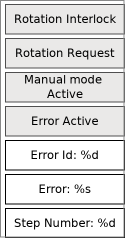
VISUALIZATION vTableBaseStationInfo  // 125x238
VAR_IN_OUT
	fbStation:FB_BaseStation;
END_VAR
    Rectangle (5,38 120x30), "Rotation Request", colour toggle: fbStation.bRotationRequest
    Rectangle (5,4 120x30), "Rotation Interlock", colour toggle: fbStation.bRotationInterlock
    Rectangle (5,106 120x30), "Error Active", colour toggle: fbStation.bError
    Rectangle (5,72 120x30), "Manual mode Active", colour toggle: fbStation.bManualModeActive
    Rectangle (5,140 120x30), "Error Id: %d", text variable: fbStation.udiErrorNumber
    Rectangle (5,208 120x30), "Step Number: %d", text variable: fbStation.iWorkStep
    Rectangle (5,174 120x30), "Error: %s", text variable: TO_STRING(fbStation.nActEvent)
END_VISUALIZATION

(* stored: Version 1.1.0.1, ProductVersion 3.1.4024.15
   Visu vTableBaseStationInfo: Id {0f14249e-ec54-4f5e-86f7-509bf5a6e481} *)
